ABB RobotStudio station: 纯净练习工作站_20210604-114951.rspag

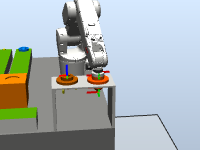
--- station ---
Station Station (saved by RobotStudio 6.4.7206.1027)
Controller System1, task T_ROB1: task frame (RAPID world) sits at (0, -189.91, 800) mm in the station
Controller System1
  mechanical unit ROB_1: IRB1200_5_90_STD_02, 6 joints, base frame (0, 0, 0) mm
Layout (positions relative to the parent item):
  - IRB1200_5_90_STD_02 [mechanism, from Robots\IRB1200_5_90_STD_02.rslib] at (0, -189.91, 800) mm; joint values [1.7401, 0.8984, -0.2519, 0, 0.9243, 1.7401] (rad or m)
  - 装配台 [part]
  - 部件 [part] at (-223.98, -561.16, 0) mm
  - 部件_2 [part] at (0, -203.49, 0) mm
  - 部件_3 [part] at (-693.25, 1032.81, 0) mm
  - 部件_4 [part] at (1137.19, 901.79, 0) mm, rotated rx 0 ry 0 rz -90 deg
  - 部件_5 [part] at (943.53, 901.79, 0) mm, rotated rx 0 ry 0 rz -90 deg
  - 零件1 [part] at (456.45, -824.42, 900.36) mm
  - 零件2 [part] at (649, -852.3, 901.96) mm
  - 爪子 [mechanism] at (-523.98, 535.35, 62.06) mm; joint values [0.02, 0.02, 0.02] (rad or m)
      links: L1, L2, L3, L4
  - 工具母头组件 [smart component] at (-123.98, 535.35, 1158) mm, rotated rx 180 ry 0 rz 180 deg
      signals: DI qijin
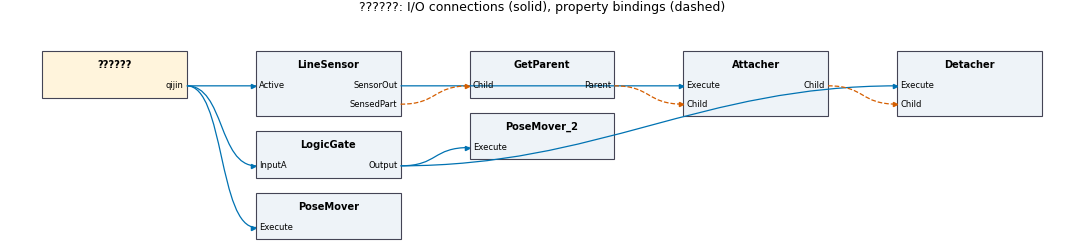
      connections:
        工具母头组件.qijin -> LineSensor.Active
        LineSensor.SensorOut -> Attacher.Execute
        工具母头组件.qijin -> LogicGate.InputA
        LogicGate.Output -> Detacher.Execute
        工具母头组件.qijin -> PoseMover.Execute
        LogicGate.Output -> PoseMover_2.Execute
        Attacher.Child => Detacher.Child
        LineSensor.SensedPart => GetParent.Child
        GetParent.Parent => Attacher.Child
    - 工具母头 [mechanism] at (600, 0, 1100.94) mm, rotated rx 180 ry 0 rz 180 deg; joint values [0, 0] (rad or m)
        TCP changtool at (0, 0, -20) mm
        TCP xipan at (0, 0, -140) mm
        TCP jiazhua at (0, 0, -106) mm
        links: L1, L2, L3
    - Attacher [smart component, from Components\Attacher.rslib] at (600, 0, 1100.94) mm, rotated rx 180 ry 0 rz 180 deg
        properties: Parent=工具母头; Flange=0; Child=爪子; Mount=false; Offset=[0 0 0]; Orientation=[0 0 0]
    - Detacher [smart component, from Components\Detacher.rslib] at (600, 0, 1100.94) mm, rotated rx 180 ry 0 rz 180 deg
        properties: Child=爪子; KeepPosition=true
    - LineSensor [smart component, from Components\LineSensor.rslib] at (600, 0, 1100.94) mm, rotated rx 180 ry 0 rz 180 deg
        properties: Start=[0.6 0 1.07794]; End=[0.6 0 1.03794]; Radius=0.002; SensedPart=L1; SensedPoint=[0.0760200042724609 0.535349975585938 1.113]
      - _sensorPart_ [part]
    - LogicGate [smart component, from Components\LogicGate.rslib] at (600, 0, 1100.94) mm, rotated rx 180 ry 0 rz 180 deg
        properties: Operator=NOT; Delay=0
    - PoseMover [smart component, from Components\PoseMover.rslib] at (600, 0, 1100.94) mm, rotated rx 180 ry 0 rz 180 deg
        properties: Mechanism=工具母头; Pose=2; Duration=0
    - PoseMover_2 [smart component, from Components\PoseMover.rslib] at (600, 0, 1100.94) mm, rotated rx 180 ry 0 rz 180 deg
        properties: Mechanism=工具母头; Pose=0; Duration=0
    - GetParent [smart component, from Components\GetParent.rslib]
        properties: Child=L1; Parent=爪子
  - 吸盘 [graphiccomponentgroup]
    - 吸盘 [part] at (-123.98, 535.34, 788.76) mm
Attachment: 工具母头组件 is attached to IRB1200_5_90_STD_02 / Link6
Targets, tools, work objects and paths stored in the station and not in the controller backup, written as RAPID:
! task T_ROB1
MODULE CalibData
  PERS tooldata changtool:=[TRUE,[[0,0,19.999],[0,0,1,0]],[1,[-1,0,0],[1,0,0,0],0,0,0]];
  PERS tooldata xipan:=[TRUE,[[0,0,140],[0,0,1,0]],[1,[-1,0,0],[1,0,0,0],0,0,0]];
  PERS tooldata jiazhua:=[TRUE,[[0,0,105.999],[0,0,1,0]],[1,[-1,0,0],[1,0,0,0],0,0,0]];
ENDMODULE

! task T_ROB1
MODULE Module1
  CONST robtarget tool2change:=[[-123.978,725.255,337.999],[1,0,0,0],[0,0,0,0],[9E+09,9E+09,9E+09,9E+09,9E+09,9E+09]];
  CONST robtarget tool1change:=[[76.02,725.26,342.999],[1,0,0,0],[0,0,0,0],[9E+09,9E+09,9E+09,9E+09,9E+09,9E+09]];
ENDMODULE


--- Backups/System1/RAPID/TASK1/SYSMOD/LINKEDM.sys ---
%%%
  VERSION:1
  LANGUAGE:ENGLISH
%%%

MODULE LINKEDM (SYSMODULE)

! FOLLOWER
!     Name of electronically linked follower axis used by operator at teach pendent.
      PERS string l_f_axis_name{5}       :=  ["",  "", "", "", ""];

!     Name of the mechanical unit for follower axis.
      PERS string l_f_mecunt_n{5}  :=  ["", "", "", "", ""];

!     Linked follower axis number in the mechanical unit (first axis in mech. unit is number 1).
      PERS num l_f_axis_no{5}      :=  [0,          0,   0,  0,  0];

! MASTER
!     Name of the mechanical unit for linked master axis.
      PERS string l_m_mecunt_n{5} :=  ["", "", "", "", ""];

!     Linked master axis number in the mechanical unit (first axis in mech. unit is number 1).
!     See axis number table in documentation for different master mechanical units.
      PERS num l_m_axis_no{5}     :=  [0,  0,  0,  0,  0];

! POSITION OFFSET
!     The increase of the allowed offset position between the master and follower
!     positions, used when starting AUTO mode. As soon as the offset is decreased
!     the old configurated parameter is used.
!     Example: 3 => the configurated value of allowed offset is increased 3 times.
      PERS num offset_ratio{5}       :=  [10,  10,   10,  10,  10];

! SPEED RATIO
!     Speed_ratio used in AUTO and JOG modes [ very_slow   slow    normal    fast]
!     Value 1 = max allowed manual speed.
      CONST num speed_ratio {20}      := [0.01, 0.01, 0.01, 0.01, 0.01,
                                          0.05, 0.05, 0.05, 0.05, 0.05,
                                          0.20, 0.20, 0.20, 0.20, 0.20,
                                          1.00, 1.00, 1.00, 1.00, 1.00];

! STEP SIZE
!     Displacement position used in JOG mode for each activation of positive or
!     negative movement.                  [very_short    short   normal   long]
!     Unit degees or meter.
      CONST num displacement {20}     := [0.001, 0.001, 0.001, 0.001, 0.001,
                                          0.005, 0.005, 0.005, 0.005, 0.005,
                                          0.020, 0.020, 0.020, 0.020, 0.020,
                                          0.100, 0.100, 0.100, 0.100, 0.100];


!-------------------------------------------------------------
 PROC Linked_m ()
      Linked_m_exe ;
 ENDPROC
ENDMODULE

--- Backups/System1/SYSPAR/EIO.cfg ---
EIO:CFG_1.0:6:1::
#
INDUSTRIAL_NETWORK:

      -Name "DeviceNet" -Label "DeviceNet Master/Slave Network" -Address "2"

      -Name "PROFINET_Anybus" -Label "PROFINET Anybus Network"\
      -Address "0.0.0.0" -SubnetMask "0.0.0.0" -Gateway "0.0.0.0"
#
DEVICENET_INTERNAL_DEVICE:

      -Name "DN_Internal_Device" -VendorName "ABB Robotics"\
      -ProductName "DeviceNet Internal Slave Device"
#
PROFINET_INTERNAL_ANYBUS_DEVICE:

      -Name "PN_Internal_Anybus" -VendorName "ABB Robotics"\
      -ProductName "PROFINET Internal Anybus Device"
